// TIA Portal V19 export
DATA_BLOCK "FinalCut_PERS"   // DB143
// stored: MemoryReserve 100
   VAR RETAIN
      PersistentValues : "udt_FinalCut_Pers";
   END_VAR
BEGIN
   PersistentValues.Par.CutHeadReload.Pause := T#0MS;
   PersistentValues.Par.CutHeadReload.Duration := T#0MS;
   PersistentValues.Par.DrawHeadReload.Pause := T#0MS;
   PersistentValues.Par.DrawHeadReload.Duration := T#0MS;
   PersistentValues.Par.MarkHeadReload.Pause := T#0MS;
   PersistentValues.Par.MarkHeadReload.Duration := T#0MS;
   PersistentValues.Par.LockingPressure.MinPressure := 75.0;
   PersistentValues.Par.LockingPressure.WorkPressure := 80.0;
   PersistentValues.Data.Locking_WorkLs := TRUE;
END_DATA_BLOCK
